TYPE ST_SubProgramConfig :
STRUCT
	Reaction 		: INT;
	TotalTableSIze 	: DINT;
	StartIdx			: DINT;
	EndIdx			: DINT;
END_STRUCT
END_TYPE

(* stored: Version 1.1.0.1, ProductVersion 3.1.4024.9
   DUT ST_SubProgramConfig: Id {fdaa1512-d575-48a5-8385-8d1124bc6738} *)
